// TIA Portal V20 export
TYPE "ScaVal_Raw"
   STRUCT
      High : DInt := 32767;   // High Value
      Low : DInt := -32768;   // Low Value
   END_STRUCT;
END_TYPE
